(* IEC 61131-3 sources: _TiaPortal14/TEST_SCL_Labor_Linearachse/Linearachse/net5.0-windows/ConfigTests/Motorschaltungen_1_3, 1 file *)

(* ---- testProgramm.st ---- *)
FUNCTION_BLOCK TestProgramm
VAR_INPUT
END_VAR
VAR_OUTPUT
END_VAR
VAR
END_VAR

(*  *********************************************************** *)
(*  Linearachse: Motorschaltungen 1 - Version 3                 *)
(*  *********************************************************** *)

IF "DigInput".S1 AND "DigInput".S2 AND "DigInput".S9 AND "DigInput".S10 THEN
    "DigOutput".P4 := true;
END_IF;

IF NOT "DigInput".S2 OR NOT "DigInput".S9 OR NOT "DigInput".S10 THEN
    "DigOutput".P4 := FALSE;
END_IF;

"DigOutput".P3 := NOT "DigInput".S9 OR NOT "DigInput".S10;

"DigOutput".P2 := NOT "DigOutput".P3 AND NOT "DigOutput".P4;
